TYPE E_HeatingState :
(
	eHeatingState_none := 0,
	eHeatingState_on,
	eHeatingState_off
);
END_TYPE

(* stored: Version 1.1.0.1
   DUT E_HeatingState: Id {a6ca2de5-2572-483c-a5a5-bb395b9da699} *)
